Staubli VAL3: removePart.pgx

public program removePart()
begin
  setMutex(bLockQueueAcces)
  //
  if bAnd(cfg:nLog,cfg:nLOGMOTION)==cfg:nLOGMOTION
    ? sConvNum+"(removePart)>>Request to remove object @ position "+toString("",nIdxPull)+" Push: "+toString("",nIdxPush)
  endIf
  //
  if nIdxPull!=nIdxPush
    call releaseObject(nIdxPull)
    nIdxPull=(nIdxPull+1)%nBufferSize
  endIf
  //
  bLockQueueAcces=false
end
